Fanuc TP program (LS listing): chwytak2.ls

/PROG  CHWYTAK2	  Macro
/ATTR
OWNER		= MNEDITOR;
COMMENT		= "";
PROG_SIZE	= 152;
CREATE		= DATE 16-10-27  TIME 10:41:00;
MODIFIED	= DATE 17-02-06  TIME 09:34:04;
FILE_NAME	= ;
VERSION		= 0;
LINE_COUNT	= 1;
MEMORY_SIZE	= 520;
PROTECT		= READ_WRITE;
TCD:  STACK_SIZE	= 0,
      TASK_PRIORITY	= 50,
      TIME_SLICE	= 0,
      BUSY_LAMP_OFF	= 0,
      ABORT_REQUEST	= 0,
      PAUSE_REQUEST	= 0;
DEFAULT_GROUP	= *,*,*,*,*;
CONTROL_CODE	= 00000000 00000000;
/APPL
/MN
   1:  RO[3:otworz chwytak 2]=(!RO[3:otworz chwytak 2]) ;
/POS
/END
